Fanuc KAREL source: kt00508.KL

-- PROVISIONAL review KL for V1013-1; original PC SHA256 696bae452438b6c66e9b4ef98afebcb699f293c09ee596760d9bebb0c6f654c8
-- Incomplete behavior may be omitted. Consult companion uncertainty JSON. Do not deploy.
PROGRAM KT00508
%NOLOCKGROUP
VAR
  OUT : BOOLEAN
-- UNRESOLVED_DECL P1 type=000102
-- UNRESOLVED_DECL P2 type=000199
BEGIN
  -- UNRESOLVED_PC offsets 5-20; opcodes 2E,22,32,35
  -- UNRESOLVED_PC offsets 25-58; opcodes 49,7E,49,7E,AC,23
  -- UNRESOLVED_PC offsets 63-67; opcodes 7F
END KT00508
